ADAPTER PortAdapter (* Adapter Interface *)
  (* Standard: 61499-1; Description: Copyright (c) 2020, 2022 Jonathan Lainer This program and the accompanying materials are made available under the terms of the Eclipse Public License 2.0 which is available at https://www.eclipse.org/legal/epl-2.0/ SPDX-License-Identifier: EPL-2.0 *)
  (* Version 0.1, 2020-03-13, Jonathan Lainer, 4DIAC-Consortium, Initial Contribution *)
  (* Compiler header: package fb.test; *)
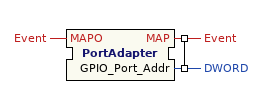
  EVENT_INPUT
    MAPO; (* Confirm Mapping *)
  END_EVENT
  EVENT_OUTPUT
    MAP WITH GPIO_Port_Addr; (* Request Mapping *)
  END_EVENT
  VAR_OUTPUT
    GPIO_Port_Addr : DWORD; (* IOMM Base Address *)
  END_VAR
  SERVICE PLUG/SOCKET (* Adapter Interface *)
    SEQUENCE request_confirm
      SOCKET.REQ(REQD) -> PLUG.REQ(REQD);
      PLUG.CNF(CNFD) -> SOCKET.CNF(CNFD);
    END_SEQUENCE
    SEQUENCE indication_response
      PLUG.IND(INDD) -> SOCKET.IND(INDD);
      SOCKET.RSP(RSPD) -> PLUG.RSP(RSPD);
    END_SEQUENCE
  END_SERVICE
END_ADAPTER
